// TIA Portal project "test3Servo_4" (V15.1)

(* hardware
DEVICE "S7-1200 station_1"  S7-1200 Station
   slot 0: "Rack_0"  S7-1200 Rack  Rack  V1.0
   slot 1: "PLC_1"  CPU 1217C DC/DC/DC  6ES7 217-1AG40-0XB0  V4.1
*)

// ===== PLC "PLC_1"  CPU 1217C DC/DC/DC =====

VAR_GLOBAL   // PLC tag table "Default tag table"
   "B1_Pulse" AT %Q0.0 : Bool;
   "B3_Pulse" AT %Q0.2 : Bool;
   "B2_Pulse" AT %Q0.1 : Bool;
   "B3_Direction" AT %Q0.6 : Bool;
   "B2_Direction" AT %Q0.5 : Bool;
   "B1_Direction" AT %Q0.4 : Bool;
   "switch1" AT %I0.0 : Bool;
   "switch2" AT %I0.2 : Bool;
   "switch3" AT %I0.4 : Bool;
   "startButton" AT %M1.1 : Bool;
   "System_Byte" AT %MB0 : Byte;
   "FirstScan" AT %M0.0 : Bool;
   "DiagStatusUpdate" AT %M0.1 : Bool;
   "AlwaysTRUE" AT %M0.2 : Bool;
   "AlwaysFALSE" AT %M0.3 : Bool;
   "simulateContact" AT %M1.0 : Bool;
   "Tag_1" AT %M1.2 : Bool;
   "Tag_2" AT %M1.3 : Bool;
   "Tag_3" AT %M1.5 : Bool;
   "Tag_4" AT %M1.6 : Bool;
END_VAR

DATA_BLOCK "motor1_DB"   // DB16
{ S7_Optimized_Access := 'TRUE' }
VERSION : 0.1
   VAR
      powerEn : Bool := true;
      powerStatus : Bool;
      powerError : Bool;
      homeExecute : Bool;
      homeDone : Bool;
      homeError : Bool;
      jogBackward : Bool;
      jogForward : Bool;
      jogVelocity : Real := 2.0;
      movExecute : Bool;
      movPosition : Real;
      movVelocity : Real := 2.0;
      movDone : Bool;
      movError : Bool;
   END_VAR
BEGIN
END_DATA_BLOCK

DATA_BLOCK "motor2_DB"   // DB17
{ S7_Optimized_Access := 'TRUE' }
VERSION : 0.1
   VAR
      powerEn : Bool := true;
      powerStatus : Bool;
      powerError : Bool;
      homeExecute : Bool;
      homeDone : Bool;
      homeError : Bool;
      jogBackward : Bool;
      jogForward : Bool;
      jogVelocity : Real := 2.0;
      movExecute : Bool;
      movPosition : Real;
      movVelocity : Real := 2.0;
      movDone : Bool;
      movError : Bool;
   END_VAR
BEGIN
END_DATA_BLOCK

DATA_BLOCK "motor3_DB"   // DB18
{ S7_Optimized_Access := 'TRUE' }
VERSION : 0.1
   VAR
      powerEn : Bool := true;
      powerStatus : Bool;
      powerError : Bool;
      homeExecute : Bool;
      homeDone : Bool;
      homeError : Bool;
      jogBackward : Bool;
      jogForward : Bool;
      jogVelocity : Real := 2.0;
      movExecute : Bool;
      movPosition : Real;
      movVelocity : Real := 2.0;
      movDone : Bool;
      movError : Bool;
   END_VAR
BEGIN
END_DATA_BLOCK

DATA_BLOCK "temporary_DB"   // DB19
{ S7_Optimized_Access := 'TRUE' }
VERSION : 0.1
   VAR
      movDone : Bool;
      start : Bool;
      movDone_Pre : Bool;
      start_Pre : Bool;
   END_VAR
BEGIN
END_DATA_BLOCK

DATA_BLOCK "TCP/IP_DB"   // DB25
{ S7_Optimized_Access := 'TRUE' }
VERSION : 0.1
   VAR
      ErrorB3 : Bool;
      DoneB3 : Bool;
      ErrorB2 : Bool;
      DoneB2 : Bool;
      ErrorB1 : Bool;
      DoneB1 : Bool;
      PLC_2_Matlab : Byte := 8;
      Matlab_2_PLC : Array[0..3] of LReal;
      TCON_DONE : Bool;
      TCON_BUSY : Bool;
      TCON_ERROR : Bool;
      TDISCON_REQ : Bool;
      TDISCON_DONE : Bool;
      TDISCON_BUSY : Bool;
      TDISCON_ERROR : Bool;
      TSEND_REQ : Bool;
      TSEND_DONE : Bool;
      TSEND_BUSY : Bool;
      TSEND_ERROR : Bool;
      TRCV_EN_R : Bool;
      TRCV_NDR : Bool;
      TRCV_BUSY : Bool;
      TRCV_ERROR : Bool;
   END_VAR
BEGIN
END_DATA_BLOCK

// folder: System blocks/Program resources

DATA_BLOCK "PLC_1_Connection_DB"   // DB21
{ S7_Optimized_Access := 'TRUE' }
AUTHOR : SIMATIC
FAMILY : MC7Plus
NAME : TC_IP_v4
VERSION : 1.0
// stored: InstanceOfName TCON_IP_v4
"TCON_IP_v4"
BEGIN
   ID := 1;
   InterfaceId := 64;
   LocalPort := 2001;
   RemotePort := 2000;
   ActiveEstablished := true;
   RemoteAddress.ADDR[1] := 192;
   RemoteAddress.ADDR[2] := 168;
   RemoteAddress.ADDR[4] := 135;
END_DATA_BLOCK

DATA_BLOCK "startTimer"   // DB26
{ S7_Optimized_Access := 'TRUE' }
AUTHOR : Simatic
FAMILY : IEC
NAME : IEC_TMR
VERSION : 1.0
// stored: InstanceOfName IEC_TIMER
"IEC_TIMER"
BEGIN
END_DATA_BLOCK

DATA_BLOCK "startTimer_TSEND"   // DB27
{ S7_Optimized_Access := 'TRUE' }
AUTHOR : Simatic
FAMILY : IEC
NAME : IEC_TMR
VERSION : 1.0
// stored: InstanceOfName IEC_TIMER
"IEC_TIMER"
BEGIN
END_DATA_BLOCK

DATA_BLOCK "setHomePulse"   // DB28
{ S7_Optimized_Access := 'TRUE' }
AUTHOR : Simatic
FAMILY : IEC
NAME : IEC_TMR
VERSION : 1.0
// stored: InstanceOfName IEC_TIMER
"IEC_TIMER"
BEGIN
END_DATA_BLOCK

// folder: (top level)

DATA_BLOCK "B1"   // DB1, Motion_DB
{ S7_Optimized_Access := 'TRUE' }
AUTHOR : SIMATIC
FAMILY : BasicMC
NAME : TO_PosAx
VERSION : 5.0
// stored: InstanceOfName TO_PositioningAxis
"TO_PositioningAxis"
BEGIN
   // Axis.LengthUnitNormalized.Distance = 1005
   // Axis.DirectionOutputEnabledCU = TRUE
   // Axis.OnlinePtoModeCU = 16#0000_0002
   // Axis.SelectedChannel2EnumCU = %Q0.4
   // Axis.SelectedChannel1EnumCU = %Q0.0
   // Pulse.MinDeltaDeltaFrequencyCU = 0.004
   // Pulse.MaxDeltaDeltaFrequencyCU = 1.0E+10
   // Pulse.MinDeltaFrequencyCU = 0.005
   // Pulse.MaxDeltaFrequencyCU = 9.5E+9
   // Pulse.MinFrequencyCU = 1.0
   // Pulse.MaxFrequencyCU = 1.0E+6
   // Pulse.OutputSourceCU = 16#0000_0000
   // Axis.SelectPTO = 0
   // Axis.LengthUnit.LastDistance = 1005
END_DATA_BLOCK

DATA_BLOCK "B2"   // DB2, Motion_DB
{ S7_Optimized_Access := 'TRUE' }
AUTHOR : SIMATIC
FAMILY : BasicMC
NAME : TO_PosAx
VERSION : 5.0
// stored: InstanceOfName TO_PositioningAxis
"TO_PositioningAxis"
BEGIN
   // Axis.LengthUnitNormalized.Distance = 1005
   // Axis.DirectionOutputEnabledCU = TRUE
   // Axis.OnlinePtoModeCU = 16#0000_0002
   // Axis.SelectedChannel2EnumCU = %Q0.5
   // Axis.SelectedChannel1EnumCU = %Q0.1
   // Pulse.MinDeltaDeltaFrequencyCU = 0.004
   // Pulse.MaxDeltaDeltaFrequencyCU = 1.0E+10
   // Pulse.MinDeltaFrequencyCU = 0.005
   // Pulse.MaxDeltaFrequencyCU = 9.5E+9
   // Pulse.MinFrequencyCU = 1.0
   // Pulse.MaxFrequencyCU = 1.0E+6
   // Pulse.OutputSourceCU = 16#0000_0000
   // Axis.SelectPTO = 1
   // Axis.OnlinePtoIndexCU = 1
   // Axis.LengthUnit.LastDistance = 1005
END_DATA_BLOCK

DATA_BLOCK "B3"   // DB3, Motion_DB
{ S7_Optimized_Access := 'TRUE' }
AUTHOR : SIMATIC
FAMILY : BasicMC
NAME : TO_PosAx
VERSION : 5.0
// stored: InstanceOfName TO_PositioningAxis
"TO_PositioningAxis"
BEGIN
   // Axis.LengthUnitNormalized.Distance = 1005
   // Axis.DirectionOutputEnabledCU = TRUE
   // Axis.OnlinePtoModeCU = 16#0000_0002
   // Axis.SelectedChannel2EnumCU = %Q0.6
   // Axis.SelectedChannel1EnumCU = %Q0.2
   // Pulse.MinDeltaDeltaFrequencyCU = 0.004
   // Pulse.MaxDeltaDeltaFrequencyCU = 1.0E+10
   // Pulse.MinDeltaFrequencyCU = 0.005
   // Pulse.MaxDeltaFrequencyCU = 9.5E+9
   // Pulse.MinFrequencyCU = 1.0
   // Pulse.MaxFrequencyCU = 1.0E+6
   // Pulse.OutputSourceCU = 16#0000_0000
   // Axis.SelectPTO = 2
   // Axis.OnlinePtoIndexCU = 2
   // Axis.LengthUnit.LastDistance = 1005
END_DATA_BLOCK

ORGANIZATION_BLOCK "Main"   // OB1, LAD, ProgramCycle
TITLE = "Main Program Sweep (Cycle)"
{ S7_Optimized_Access := 'TRUE' }
VERSION : 0.1
   VAR_INPUT
      Initial_Call : Bool;   // Initial call of this OB
      Remanence : Bool;   // =True, if remanent data are available
   END_VAR
   VAR_TEMP   // added for the SCL form of the ladder/FBD networks
      _w1 : Bool;
      _w2 : Bool;
   END_VAR
BEGIN

REGION Network 1: go home
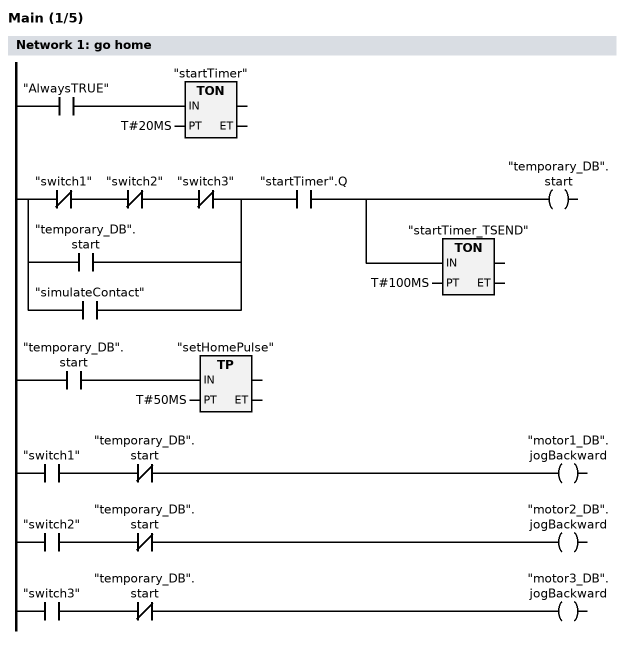
   "startTimer".TON(IN := "AlwaysTRUE", PT := T#20MS);
   "temporary_DB".start := ((NOT "switch1" AND NOT "switch2" AND NOT "switch3") OR "temporary_DB".start OR "simulateContact") AND "startTimer".Q;
   "startTimer_TSEND".TON(IN := "temporary_DB".start, PT := T#100MS);
   "setHomePulse".TP(IN := "temporary_DB".start, PT := T#50MS);
   "motor1_DB".jogBackward := "switch1" AND NOT "temporary_DB".start;
   "motor2_DB".jogBackward := "switch2" AND NOT "temporary_DB".start;
   "motor3_DB".jogBackward := "switch3" AND NOT "temporary_DB".start;
END_REGION

REGION Network 2
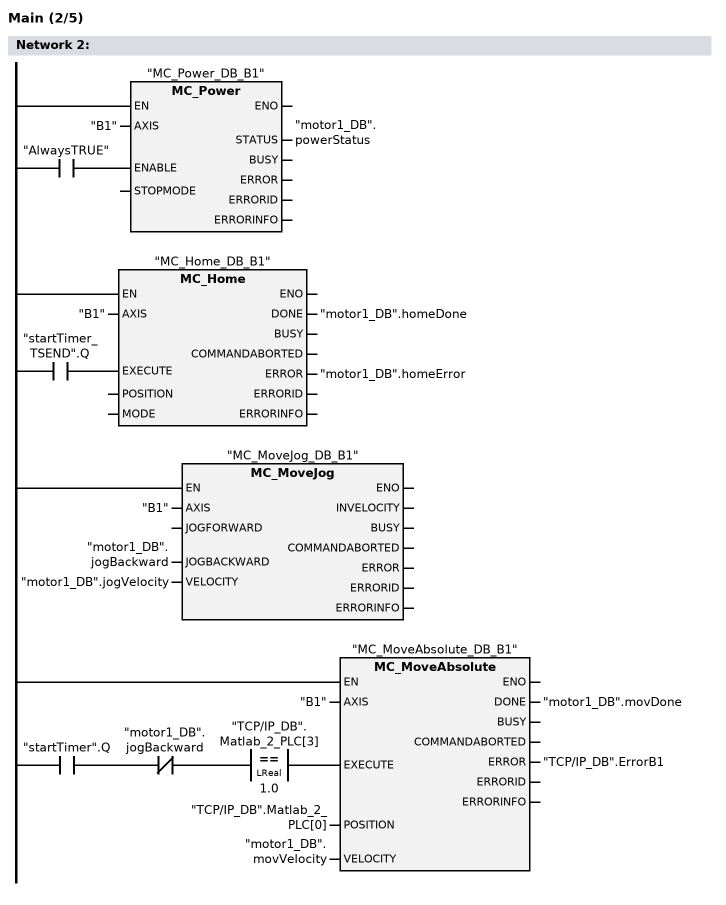
   "MC_Power_DB_B1"(Axis := "B1", Enable := "AlwaysTRUE", Status => "motor1_DB".powerStatus);   // MC_Power
   "MC_Home_DB_B1"(Axis := "B1",   // MC_Home
                   Execute := "startTimer_TSEND".Q,
                   Done => "motor1_DB".homeDone,
                   Error => "motor1_DB".homeError);
   "MC_MoveJog_DB_B1"(Axis := "B1", JogBackward := "motor1_DB".jogBackward, Velocity := "motor1_DB".jogVelocity);   // MC_MoveJog
   "MC_MoveAbsolute_DB_B1"(Axis := "B1",   // MC_MoveAbsolute
                           Execute := "startTimer".Q AND NOT "motor1_DB".jogBackward AND ("TCP/IP_DB".Matlab_2_PLC[3] = 1.0),
                           Position := "TCP/IP_DB".Matlab_2_PLC[0],
                           Velocity := "motor1_DB".movVelocity,
                           Done => "motor1_DB".movDone,
                           Error => "TCP/IP_DB".ErrorB1);
END_REGION

REGION Network 3
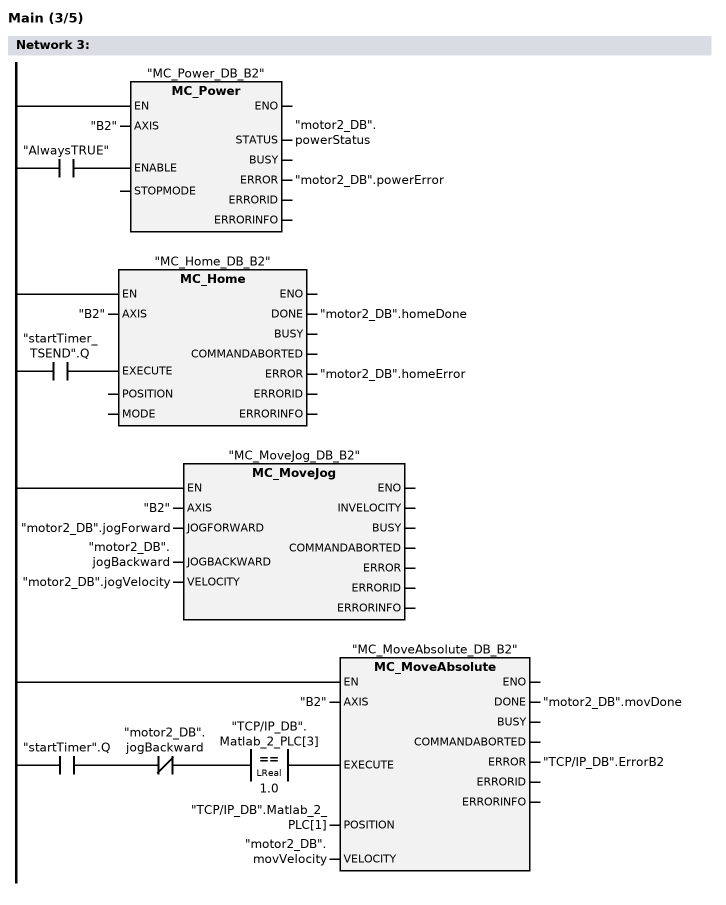
   "MC_Power_DB_B2"(Axis := "B2",   // MC_Power
                    Enable := "AlwaysTRUE",
                    Status => "motor2_DB".powerStatus,
                    Error => "motor2_DB".powerError);
   "MC_Home_DB_B2"(Axis := "B2",   // MC_Home
                   Execute := "startTimer_TSEND".Q,
                   Done => "motor2_DB".homeDone,
                   Error => "motor2_DB".homeError);
   "MC_MoveJog_DB_B2"(Axis := "B2",   // MC_MoveJog
                      JogForward := "motor2_DB".jogForward,
                      JogBackward := "motor2_DB".jogBackward,
                      Velocity := "motor2_DB".jogVelocity);
   "MC_MoveAbsolute_DB_B2"(Axis := "B2",   // MC_MoveAbsolute
                           Execute := "startTimer".Q AND NOT "motor2_DB".jogBackward AND ("TCP/IP_DB".Matlab_2_PLC[3] = 1.0),
                           Position := "TCP/IP_DB".Matlab_2_PLC[1],
                           Velocity := "motor2_DB".movVelocity,
                           Done => "motor2_DB".movDone,
                           Error => "TCP/IP_DB".ErrorB2);
END_REGION

REGION Network 4
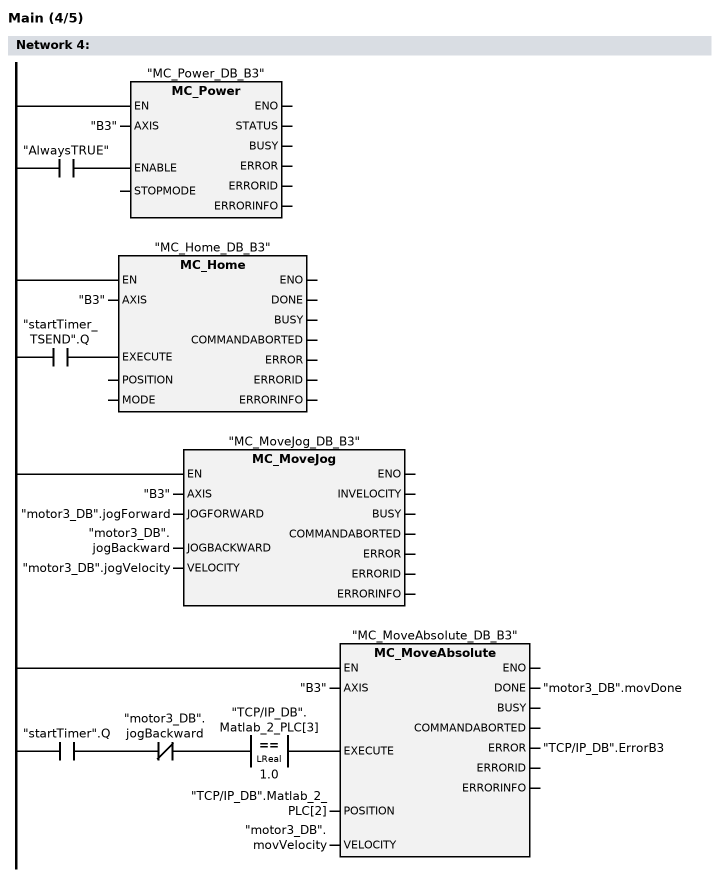
   "MC_Power_DB_B3"(Axis := "B3", Enable := "AlwaysTRUE");   // MC_Power
   "MC_Home_DB_B3"(Axis := "B3", Execute := "startTimer_TSEND".Q);   // MC_Home
   "MC_MoveJog_DB_B3"(Axis := "B3",   // MC_MoveJog
                      JogForward := "motor3_DB".jogForward,
                      JogBackward := "motor3_DB".jogBackward,
                      Velocity := "motor3_DB".jogVelocity);
   "MC_MoveAbsolute_DB_B3"(Axis := "B3",   // MC_MoveAbsolute
                           Execute := "startTimer".Q AND NOT "motor3_DB".jogBackward AND ("TCP/IP_DB".Matlab_2_PLC[3] = 1.0),
                           Position := "TCP/IP_DB".Matlab_2_PLC[2],
                           Velocity := "motor3_DB".movVelocity,
                           Done => "motor3_DB".movDone,
                           Error => "TCP/IP_DB".ErrorB3);
END_REGION

REGION Network 5: communicate with Matlab
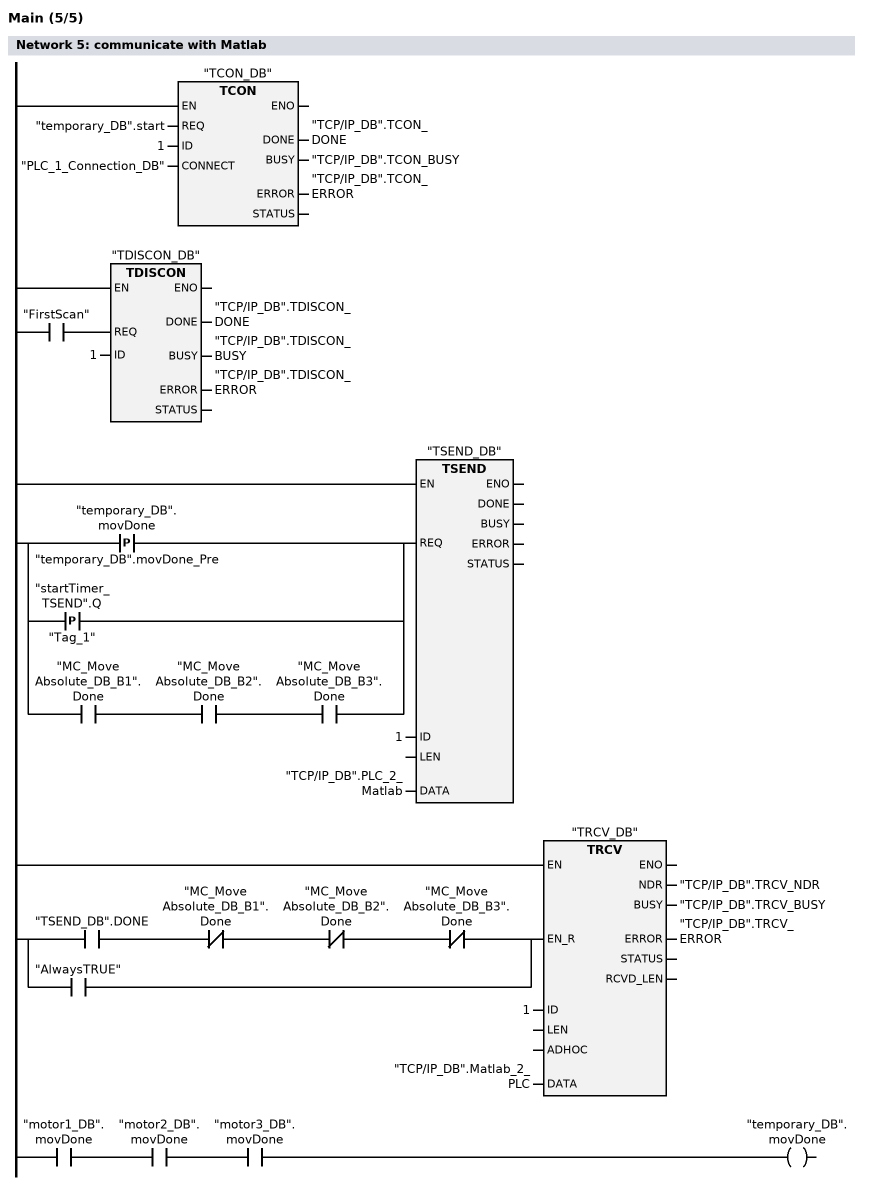
   "TCON_DB"(REQ := "temporary_DB".start,   // TCON
             ID := 1,
             CONNECT := "PLC_1_Connection_DB",
             DONE => "TCP/IP_DB".TCON_DONE,
             BUSY => "TCP/IP_DB".TCON_BUSY,
             ERROR => "TCP/IP_DB".TCON_ERROR);
   "TDISCON_DB"(REQ := "FirstScan",   // TDISCON
                ID := 1,
                DONE => "TCP/IP_DB".TDISCON_DONE,
                BUSY => "TCP/IP_DB".TDISCON_BUSY,
                ERROR => "TCP/IP_DB".TDISCON_ERROR);
   #_w1 := "temporary_DB".movDone AND NOT "temporary_DB".movDone_Pre;   // rising edge of "temporary_DB".movDone
   "temporary_DB".movDone_Pre := "temporary_DB".movDone;
   #_w2 := "startTimer_TSEND".Q AND NOT "Tag_1";   // rising edge of "startTimer_TSEND".Q
   "Tag_1" := "startTimer_TSEND".Q;
   "TSEND_DB"(REQ := #_w1 OR #_w2 OR ("MC_MoveAbsolute_DB_B1".Done AND "MC_MoveAbsolute_DB_B2".Done AND "MC_MoveAbsolute_DB_B3".Done),   // TSEND
              ID := 1,
              DATA := "TCP/IP_DB".PLC_2_Matlab);
   "TRCV_DB"(EN_R := ("TSEND_DB".DONE AND NOT "MC_MoveAbsolute_DB_B1".Done AND NOT "MC_MoveAbsolute_DB_B2".Done AND NOT "MC_MoveAbsolute_DB_B3".Done) OR "AlwaysTRUE",   // TRCV
             ID := 1,
             DATA := "TCP/IP_DB".Matlab_2_PLC,
             NDR => "TCP/IP_DB".TRCV_NDR,
             BUSY => "TCP/IP_DB".TRCV_BUSY,
             ERROR => "TCP/IP_DB".TRCV_ERROR);
   "temporary_DB".movDone := "motor1_DB".movDone AND "motor2_DB".movDone AND "motor3_DB".movDone;
END_REGION
END_ORGANIZATION_BLOCK